// TIA Portal V17 export
// export: Created 2025-03-05T08:03:46.6788071Z, ExportSetting WithDefaults, DisplayName Totally Integrated Automation Portal, DisplayVersion V17 Update 8, DisplayName TIA Portal Openness, DisplayVersion V17 Update 8, DisplayName TIA Portal Version Control Interface, DisplayVersion V17, DisplayName SINAMICS Startdrive Advanced, DisplayVersion V17 SP2, DisplayName SINAMICS Startdrive G110M, G120, G120C, G120D, G120P, G115D, DisplayVersion V17 SP2, DisplayName SINAMICS Startdrive G130, G150, S120, S150, SINAMICS MV, S210, DisplayVersion V17 SP2, DisplayName STEP 7 Professional, DisplayVersion V17 Update 8, DisplayName SINUMERIK ONE STEP 7 Toolbox, DisplayVersion V17 Update 12, DisplayName SINUMERIK 840D sl STEP 7 Toolbox, DisplayVersion V17 Update 12, DisplayName STEP 7 Safety, DisplayVersion V17 Update 6, DisplayName WinCC Advanced, DisplayVersion V17 Update 8
TYPE "GLOBAL_DATA_CLADDING"
// stored: IsFailsafeCompliant false
   STRUCT
      NO_MACHINE_CYCLE_RUN_P : Bool;   // NO CYCLE MACHINE RUN PROGRAM / NO MACHINE CYCLE RUNNING PULSE
      ANY_MACHINE_CYCLE_RUN_P : Bool;   // ANY MACHINE CYCLE RUN PROGRAM / ANY MACHINE CYCLE RUNNING PULSE
      NO_MACHINE_CYCLE_RUN_HOPPER_UNIT_01_P : Bool;   // NO CYCLE MACHINE RUN PROGRAM / NO MACHINE CYCLE RUNNING HOPPER UNIT 01 PULSE
      ANY_HOPPER_UNIT_01_CYCLE_RUN_P : Bool;   // ANY MACHINE CYCLE RUN PROGRAM / ANY HOPPER UNIT 01 CYCLE RUNNING PULSE
      NO_MACHINE_CYCLE_RUN_HOPPER_UNIT_02_P : Bool;   // NO CYCLE MACHINE RUN PROGRAM / NO MACHINE CYCLE RUNNING HOPPER UNIT 02 PULSE
      ANY_HOPPER_UNIT_02_CYCLE_RUN_P : Bool;   // ANY MACHINE CYCLE RUN PROGRAM / ANY HOPPER UNIT 02 CYCLE RUNNING PULSE
      ANY_MACHINE_CYCLE_RUN : Bool;   // ANY MACHINE CYCLE RUN / ANY MACHINE CYCLE RUNNING
      ANY_UNIT_01_CYCLE_RUN : Bool;   // ANY MACHINE CYCLE RUN / ANY UNIT 01 CYCLE RUNNING
      ANY_UNIT_02_CYCLE_RUN : Bool;   // ANY MACHINE CYCLE RUN / ANY UNIT 02 CYCLE RUNNING
      ANY_HOPPER_UNIT_01_CYCLE_RUN : Bool;   // ANY MACHINE CYCLE RUN / ANY HOPPER UNIT 01 CYCLE RUNNING
      ANY_HOPPER_UNIT_02_CYCLE_RUN : Bool;   // ANY MACHINE CYCLE RUN / ANY HOPPER UNIT 02 CYCLE RUNNING
      ANY_HOPPER_1_UNIT_01_CYCLE_RUN : Bool;   // ANY HOPPER 1 UNIT 01 CYCLE RUNNING
      ANY_HOPPER_2_UNIT_01_CYCLE_RUN : Bool;   // ANY HOPPER 2 UNIT 01 CYCLE RUNNING
      ANY_HOPPER_1_UNIT_02_CYCLE_RUN : Bool;   // ANY HOPPER 1 UNIT 02 CYCLE RUNNING
      ANY_HOPPER_2_UNIT_02_CYCLE_RUN : Bool;   // ANY HOPPER 2 UNIT 02 CYCLE RUNNING
      ANY_HOPPER_3_UNIT_02_CYCLE_RUN : Bool;   // ANY HOPPER 3 UNIT 02 CYCLE RUNNING
      ANY_POWDER_FEEDER_RUN : Bool;   // ANY POWDER FEEDER RUNNING
      AUX0 : Bool;   // AUXILIARY 0
      AUX1 : Bool;   // AUXILIARY 1
      AUX2 : Bool;   // AUXILIARY 2
      AUX3 : Bool;   // AUXILIARY 3
      AUX4 : Bool;   // AUXILIARY 4
      AUX5 : Bool;   // AUXILIARY 5
      AUX6 : Bool;   // AUXILIARY 6
      AUX7 : Bool;   // AUXILIARY 7
      AUX8 : Bool;   // AUXILIARY 7
      AUX9 : Bool;   // AUXILIARY 7
      AUX10 : Bool;   // AUXILIARY 7
      AUX11 : Bool;   // AUXILIARY 7
   END_STRUCT;
END_TYPE
